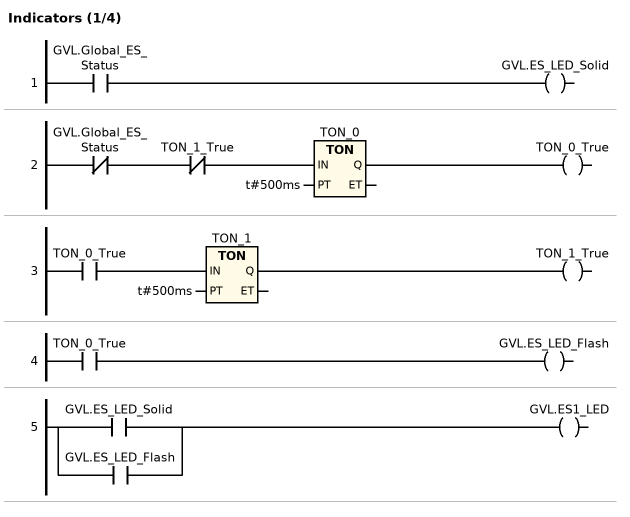
// NETWORK 1
GVL.ES_LED_Solid := GVL.Global_ES_Status;

// NETWORK 2
TON_0(IN := NOT GVL.Global_ES_Status AND NOT TON_1_True, PT := t#500ms); // TON
TON_0_True := TON_0.Q;

// NETWORK 3
TON_1(IN := TON_0_True, PT := t#500ms); // TON
TON_1_True := TON_1.Q;

// NETWORK 4
GVL.ES_LED_Flash := TON_0_True;

// NETWORK 5
GVL.ES1_LED := GVL.ES_LED_Solid OR GVL.ES_LED_Flash;

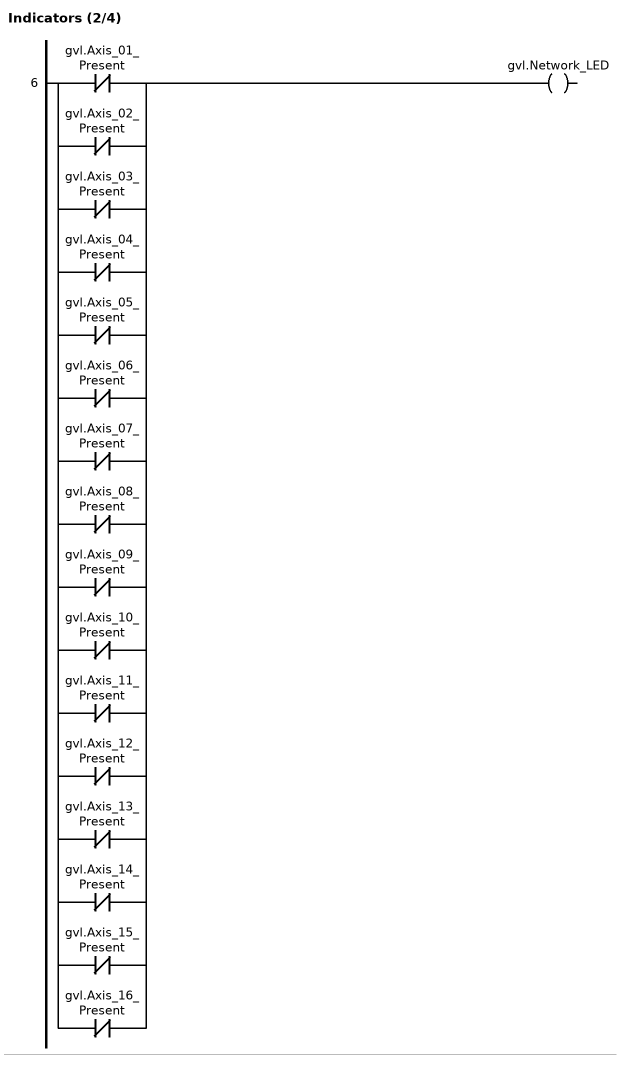
// NETWORK 6
gvl.Network_LED := NOT gvl.Axis_01_Present OR NOT gvl.Axis_02_Present OR NOT gvl.Axis_03_Present OR NOT gvl.Axis_04_Present OR NOT gvl.Axis_05_Present OR NOT gvl.Axis_06_Present OR NOT gvl.Axis_07_Present OR NOT gvl.Axis_08_Present OR NOT gvl.Axis_09_Present OR NOT gvl.Axis_10_Present OR NOT gvl.Axis_11_Present OR NOT gvl.Axis_12_Present OR NOT gvl.Axis_13_Present OR NOT gvl.Axis_14_Present OR NOT gvl.Axis_15_Present OR NOT gvl.Axis_16_Present;

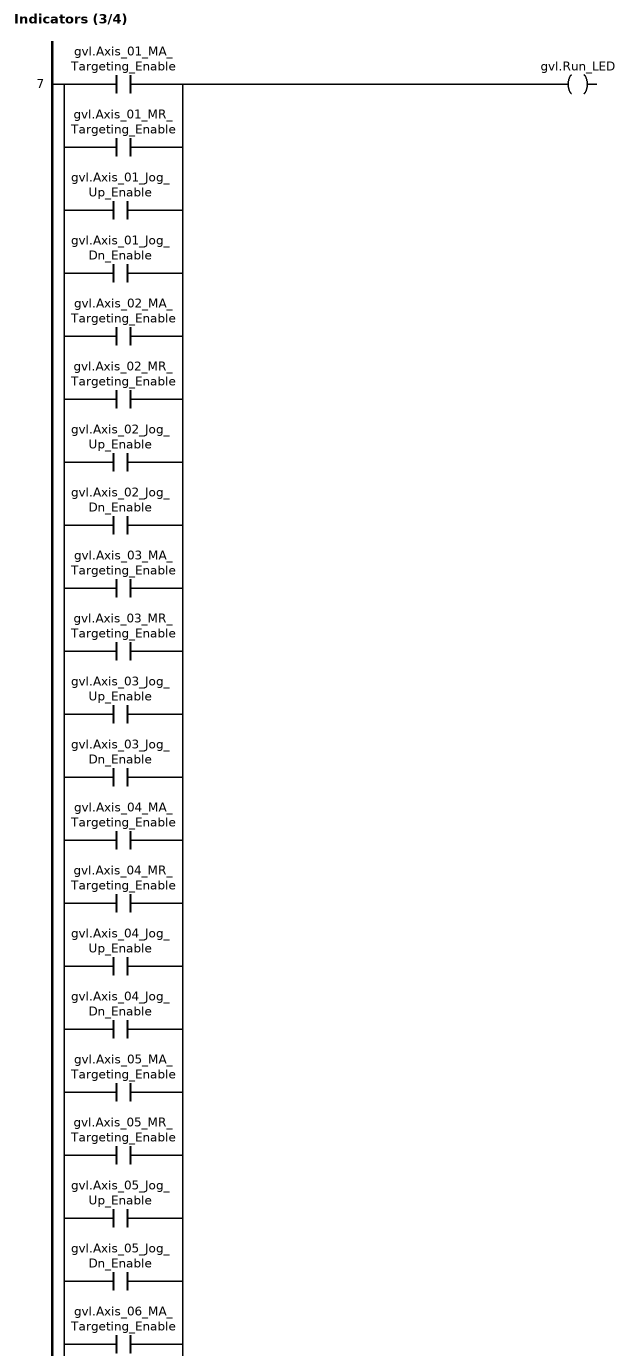
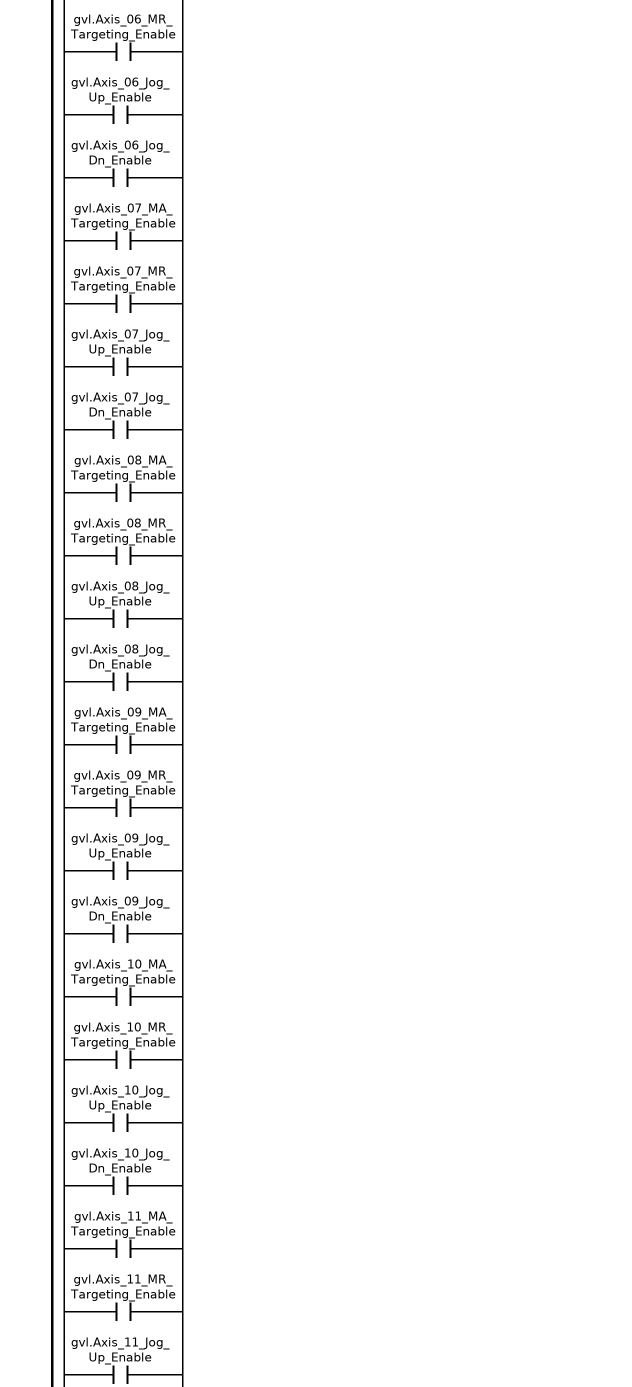
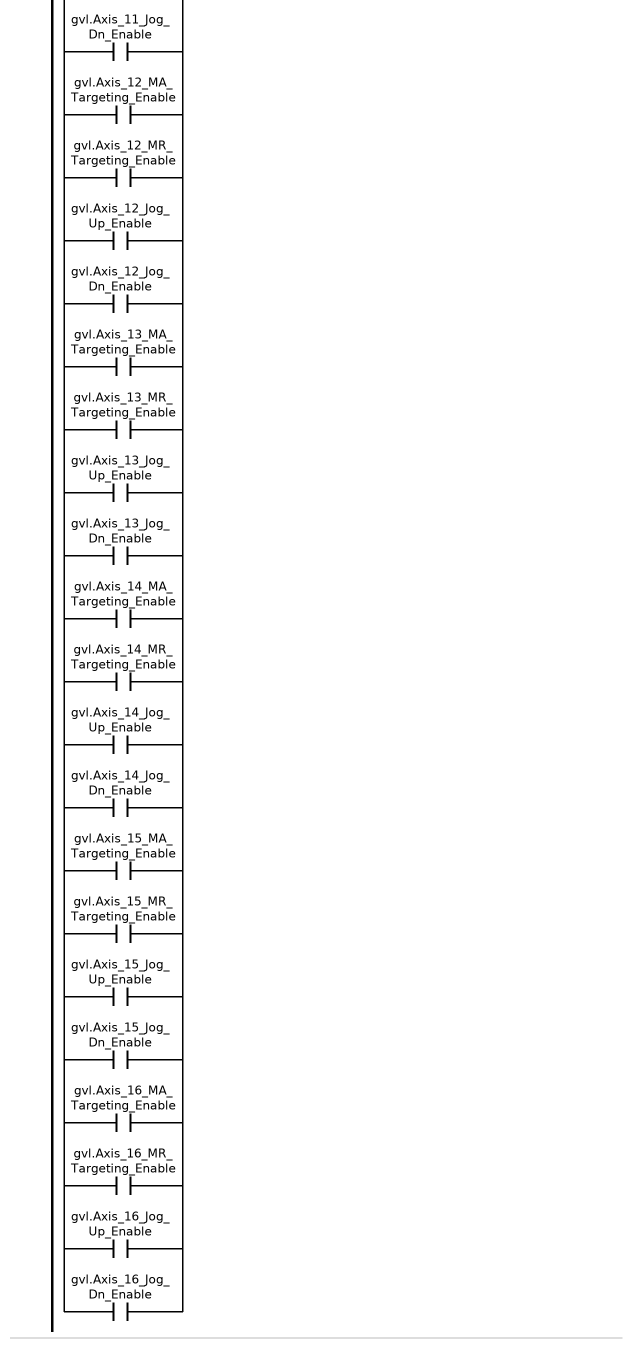
// NETWORK 7
gvl.Run_LED := gvl.Axis_01_MA_Targeting_Enable OR gvl.Axis_01_MR_Targeting_Enable OR gvl.Axis_01_Jog_Up_Enable OR gvl.Axis_01_Jog_Dn_Enable OR gvl.Axis_02_MA_Targeting_Enable OR gvl.Axis_02_MR_Targeting_Enable OR gvl.Axis_02_Jog_Up_Enable OR gvl.Axis_02_Jog_Dn_Enable OR gvl.Axis_03_MA_Targeting_Enable OR gvl.Axis_03_MR_Targeting_Enable OR gvl.Axis_03_Jog_Up_Enable OR gvl.Axis_03_Jog_Dn_Enable OR gvl.Axis_04_MA_Targeting_Enable OR gvl.Axis_04_MR_Targeting_Enable OR gvl.Axis_04_Jog_Up_Enable OR gvl.Axis_04_Jog_Dn_Enable OR gvl.Axis_05_MA_Targeting_Enable OR gvl.Axis_05_MR_Targeting_Enable OR gvl.Axis_05_Jog_Up_Enable OR gvl.Axis_05_Jog_Dn_Enable OR gvl.Axis_06_MA_Targeting_Enable OR gvl.Axis_06_MR_Targeting_Enable OR gvl.Axis_06_Jog_Up_Enable OR gvl.Axis_06_Jog_Dn_Enable OR gvl.Axis_07_MA_Targeting_Enable OR gvl.Axis_07_MR_Targeting_Enable OR gvl.Axis_07_Jog_Up_Enable OR gvl.Axis_07_Jog_Dn_Enable OR gvl.Axis_08_MA_Targeting_Enable OR gvl.Axis_08_MR_Targeting_Enable OR gvl.Axis_08_Jog_Up_Enable OR gvl.Axis_08_Jog_Dn_Enable OR gvl.Axis_09_MA_Targeting_Enable OR gvl.Axis_09_MR_Targeting_Enable OR gvl.Axis_09_Jog_Up_Enable OR gvl.Axis_09_Jog_Dn_Enable OR gvl.Axis_10_MA_Targeting_Enable OR gvl.Axis_10_MR_Targeting_Enable OR gvl.Axis_10_Jog_Up_Enable OR gvl.Axis_10_Jog_Dn_Enable OR gvl.Axis_11_MA_Targeting_Enable OR gvl.Axis_11_MR_Targeting_Enable OR gvl.Axis_11_Jog_Up_Enable OR gvl.Axis_11_Jog_Dn_Enable OR gvl.Axis_12_MA_Targeting_Enable OR gvl.Axis_12_MR_Targeting_Enable OR gvl.Axis_12_Jog_Up_Enable OR gvl.Axis_12_Jog_Dn_Enable OR gvl.Axis_13_MA_Targeting_Enable OR gvl.Axis_13_MR_Targeting_Enable OR gvl.Axis_13_Jog_Up_Enable OR gvl.Axis_13_Jog_Dn_Enable OR gvl.Axis_14_MA_Targeting_Enable OR gvl.Axis_14_MR_Targeting_Enable OR gvl.Axis_14_Jog_Up_Enable OR gvl.Axis_14_Jog_Dn_Enable OR gvl.Axis_15_MA_Targeting_Enable OR gvl.Axis_15_MR_Targeting_Enable OR gvl.Axis_15_Jog_Up_Enable OR gvl.Axis_15_Jog_Dn_Enable OR gvl.Axis_16_MA_Targeting_Enable OR gvl.Axis_16_MR_Targeting_Enable OR gvl.Axis_16_Jog_Up_Enable OR gvl.Axis_16_Jog_Dn_Enable;

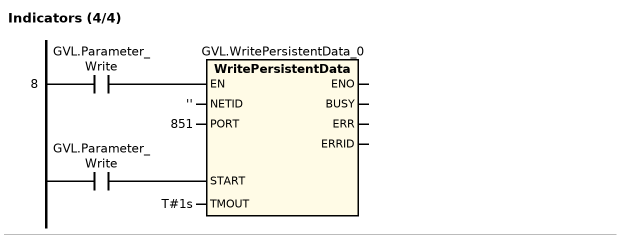
// NETWORK 8
IF GVL.Parameter_Write THEN
    GVL.WritePersistentData_0(NETID := '', PORT := 851, START := GVL.Parameter_Write, TMOUT := T#1s); // WritePersistentData
END_IF

END_PROGRAM

// ---- POUs/UIFB.TcPOU
FUNCTION_BLOCK FINAL UIFB
VAR_INPUT
END_VAR
VAR_OUTPUT
END_VAR
VAR
END_VAR

{attribute 'TcRpcEnable'}
METHOD PUBLIC ClearMotionAndJog : DINT
GVL.Axis_01_MA_Enable := GVL.Axis_01_MR_Enable := GVL.Axis_01_Jog_Up_Enable := GVL.Axis_01_Jog_Dn_Enable := 
GVL.Axis_02_MA_Enable := GVL.Axis_02_MR_Enable := GVL.Axis_02_Jog_Up_Enable := GVL.Axis_02_Jog_Dn_Enable := 
GVL.Axis_03_MA_Enable := GVL.Axis_03_MR_Enable := GVL.Axis_03_Jog_Up_Enable := GVL.Axis_03_Jog_Dn_Enable := 
GVL.Axis_04_MA_Enable := GVL.Axis_04_MR_Enable := GVL.Axis_04_Jog_Up_Enable := GVL.Axis_04_Jog_Dn_Enable := 
GVL.Axis_05_MA_Enable := GVL.Axis_05_MR_Enable := GVL.Axis_05_Jog_Up_Enable := GVL.Axis_05_Jog_Dn_Enable := 
GVL.Axis_06_MA_Enable := GVL.Axis_06_MR_Enable := GVL.Axis_06_Jog_Up_Enable := GVL.Axis_06_Jog_Dn_Enable := 
GVL.Axis_07_MA_Enable := GVL.Axis_07_MR_Enable := GVL.Axis_07_Jog_Up_Enable := GVL.Axis_07_Jog_Dn_Enable := 
GVL.Axis_08_MA_Enable := GVL.Axis_08_MR_Enable := GVL.Axis_08_Jog_Up_Enable := GVL.Axis_08_Jog_Dn_Enable := 
GVL.Axis_09_MA_Enable := GVL.Axis_09_MR_Enable := GVL.Axis_09_Jog_Up_Enable := GVL.Axis_09_Jog_Dn_Enable := 
GVL.Axis_10_MA_Enable := GVL.Axis_10_MR_Enable := GVL.Axis_10_Jog_Up_Enable := GVL.Axis_10_Jog_Dn_Enable := 
GVL.Axis_11_MA_Enable := GVL.Axis_11_MR_Enable := GVL.Axis_11_Jog_Up_Enable := GVL.Axis_11_Jog_Dn_Enable := 
GVL.Axis_12_MA_Enable := GVL.Axis_12_MR_Enable := GVL.Axis_12_Jog_Up_Enable := GVL.Axis_12_Jog_Dn_Enable := 
GVL.Axis_13_MA_Enable := GVL.Axis_13_MR_Enable := GVL.Axis_13_Jog_Up_Enable := GVL.Axis_13_Jog_Dn_Enable := 
GVL.Axis_14_MA_Enable := GVL.Axis_14_MR_Enable := GVL.Axis_14_Jog_Up_Enable := GVL.Axis_14_Jog_Dn_Enable := 
GVL.Axis_15_MA_Enable := GVL.Axis_15_MR_Enable := GVL.Axis_15_Jog_Up_Enable := GVL.Axis_15_Jog_Dn_Enable := 
GVL.Axis_16_MA_Enable := GVL.Axis_16_MR_Enable := GVL.Axis_16_Jog_Up_Enable := GVL.Axis_16_Jog_Dn_Enable := 
GVL.Axis_17_MA_Enable := GVL.Axis_17_MR_Enable := GVL.Axis_17_Jog_Up_Enable := GVL.Axis_17_Jog_Dn_Enable := 
GVL.Axis_18_MA_Enable := GVL.Axis_18_MR_Enable := GVL.Axis_18_Jog_Up_Enable := GVL.Axis_18_Jog_Dn_Enable := 
GVL.Axis_19_MA_Enable := GVL.Axis_19_MR_Enable := GVL.Axis_19_Jog_Up_Enable := GVL.Axis_19_Jog_Dn_Enable := 
GVL.Axis_20_MA_Enable := GVL.Axis_20_MR_Enable := GVL.Axis_20_Jog_Up_Enable := GVL.Axis_20_Jog_Dn_Enable := 
GVL.Axis_21_MA_Enable := GVL.Axis_21_MR_Enable := GVL.Axis_21_Jog_Up_Enable := GVL.Axis_21_Jog_Dn_Enable := 
GVL.Axis_22_MA_Enable := GVL.Axis_22_MR_Enable := GVL.Axis_22_Jog_Up_Enable := GVL.Axis_22_Jog_Dn_Enable := 
GVL.Axis_23_MA_Enable := GVL.Axis_23_MR_Enable := GVL.Axis_23_Jog_Up_Enable := GVL.Axis_23_Jog_Dn_Enable := 
GVL.Axis_24_MA_Enable := GVL.Axis_24_MR_Enable := GVL.Axis_24_Jog_Up_Enable := GVL.Axis_24_Jog_Dn_Enable := 
0;

ClearMotionAndJog := 0;
END_METHOD

{attribute 'TcRpcEnable'}
METHOD PUBLIC GetMotorsGroup : DINT
VAR_OUTPUT
	res: ARRAY[0..15] OF INT;
END_VAR
VAR
	ptr: POINTER TO BOOL;
	im, ig:INT;
END_VAR
ptr := ADR(GVL.Group_01_Axis_01);
MEMSET(destAddr:=ADR(res[0]), fillByte:=0, n:=SIZEOF(res));
FOR ig := 1 TO 8 DO
	FOR im := 0 TO 15 DO
		IF ptr^ THEN
			IF res[im] <> 0 THEN
				ptr^ := 0;
			ELSE
				res[im] := ig;
			END_IF
		END_IF
		ptr := ptr + 1;
	END_FOR
END_FOR

GetMotorsGroup := 0;
RETURN;
END_METHOD

{attribute 'TcRpcEnable'}
METHOD PUBLIC SaveGroupMotors : DINT
VAR_INPUT
	Group:INT;
	Bitmap:WORD;
END_VAR
VAR
	ptr: POINTER TO BOOL;
	i:INT;
END_VAR
ptr := ADR(GVL.Group_01_Axis_01) + Group * 16;

FOR i := 0 TO 15 DO
	ptr^ := (Bitmap AND 1) <> 0;
	ptr := ptr + 1;
	Bitmap := SHR(Bitmap, 1);
END_FOR

SaveGroupMotors := 0;
RETURN;
END_METHOD

END_FUNCTION_BLOCK

// ---- POUs/CheckDivDInt.TcPOU
// Implicitly generated code : DO NOT EDIT
FUNCTION CheckDivDInt : DINT
VAR_INPUT
	divisor:DINT;
END_VAR

// Implicitly generated code : Only an Implementation suggestion
{noflow}
IF divisor = 0 THEN
	CheckDivDInt:=1;
ELSE
	CheckDivDInt:=divisor;
END_IF;
{flow}

END_FUNCTION

// ---- POUs/CheckDivLInt.TcPOU
// Implicitly generated code : DO NOT EDIT
FUNCTION CheckDivLInt : LINT
VAR_INPUT
	divisor:LINT;
END_VAR

// Implicitly generated code : Only an Implementation suggestion
{noflow}
IF divisor = 0 THEN
	CheckDivLInt:=1;
ELSE
	CheckDivLInt:=divisor;
END_IF;
{flow}

END_FUNCTION

// ---- POUs/CheckDivLReal.TcPOU
// Implicitly generated code : DO NOT EDIT
FUNCTION CheckDivLReal : LREAL
VAR_INPUT
	divisor:LREAL;
END_VAR

// Implicitly generated code : Only an Implementation suggestion
{noflow}
IF divisor = 0 THEN
	CheckDivLReal:=1;
ELSE
	CheckDivLReal:=divisor;
END_IF;
{flow}

END_FUNCTION

// ---- POUs/CheckDivReal.TcPOU
// Implicitly generated code : DO NOT EDIT
FUNCTION CheckDivReal : REAL
VAR_INPUT
	divisor:REAL;
END_VAR

// Implicitly generated code : Only an Implementation suggestion
{noflow}
IF divisor = 0 THEN
	CheckDivReal:=1;
ELSE
	CheckDivReal:=divisor;
END_IF;
{flow}

END_FUNCTION
